// TIA Portal V17 export
// export: Created 2025-06-26T06:49:21.3533278Z, ExportSetting WithDefaults, DisplayName Totally Integrated Automation Portal, DisplayVersion V17 Update 8, DisplayName TIA Portal Openness, DisplayVersion V17 Update 8, DisplayName TIA Portal Version Control Interface, DisplayVersion V17, DisplayName STEP 7 Professional, DisplayVersion V17 Update 8, DisplayName STEP 7 Safety, DisplayVersion V17 Update 6, DisplayName WinCC Advanced, DisplayVersion V17 Update 8
DATA_BLOCK "Modbus_Comm_Load_DB"   // DB12
// stored: AutoNumber true, DBAccessibleFromOPCUA true, InstanceOfName Modbus_Comm_Load, OfSystemLibElement Modbus_Comm_Load, OfSystemLibVersion 5.0
"Modbus_Comm_Load"
   // VAR_INPUT
   //    REQ : Bool;
   //    PORT : PORT;
   //    BAUD : UDInt;
   //    PARITY : UInt;
   //    FLOW_CTRL : UInt;
   //    RTS_ON_DLY : UInt;
   //    RTS_OFF_DLY : UInt;
   //    RESP_TO : UInt;
   // END_VAR
   // VAR_OUTPUT
   //    DONE : Bool;
   //    ERROR : Bool;
   //    STATUS : Word;
   // END_VAR
   // VAR_IN_OUT
   //    MB_DB : P2P_MB_BASE;
   // END_VAR
   // VAR
   //    ICHAR_GAP : Word;
   //    RETRIES : Word;
   //    MODE : USInt;
   //    LINE_PRE : USInt;
   //    BRK_DET : USInt;
   //    EN_DIAG_ALARM : Bool;
   //    STOP_BITS : USInt;
   //    EN_SUPPLY_VOLT : Bool;
   //    b_e_REQ : Bool;
   //    y_state : SInt;
   //    Send_Config { S7_SetPoint := 'True'} : Send_Config;
   //    Receive_Config { S7_SetPoint := 'True'} : Receive_Config;
   //    Receive_Conditions { S7_SetPoint := 'True'} : Receive_Conditions;
   //    WRREC { S7_SetPoint := 'True'} : WRREC;
   //    RDREC { S7_SetPoint := 'True'} : RDREC;
   //    port_w_record { ExternalVisible := 'False'; S7_SetPoint := 'True'} : P2P_MB_PortData;
   //    err_record { ExternalVisible := 'False'; S7_SetPoint := 'True'} : P2P_RdEstat;
   //    ftrs_w_record { ExternalVisible := 'False'; S7_SetPoint := 'True'} : P2P_FeaturesData;
   //    wlen : UInt;
   // END_VAR
BEGIN
END_DATA_BLOCK
